// Mitsubishi GX Works2 project: PARKING   PLC: FX1S
// PARKING

PROGRAM MAIN
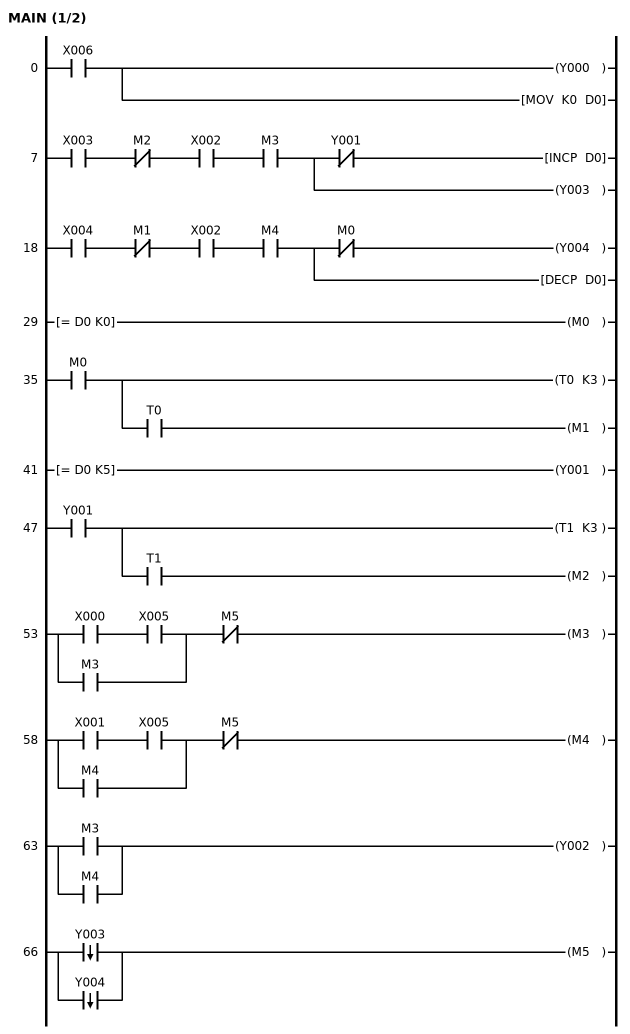
0     LD      X006
      OUT     Y000
      MOV     K0 D0
7     LD      X003
      ANI     M2
      AND     X002
      AND     M3
      MPS
      ANI     Y001
      INCP    D0
      MPP
      OUT     Y003
18    LD      X004
      ANI     M1
      AND     X002
      AND     M4
      MPS
      ANI     M0
      OUT     Y004
      MPP
      DECP    D0
29    LD=     D0 K0
      OUT     M0
35    LD      M0
      OUT     T0 K3
      AND     T0
      OUT     M1
41    LD=     D0 K5
      OUT     Y001
47    LD      Y001
      OUT     T1 K3
      AND     T1
      OUT     M2
53    LD      X000
      AND     X005
      OR      M3
      ANI     M5
      OUT     M3
58    LD      X001
      AND     X005
      OR      M4
      ANI     M5
      OUT     M4
63    LD      M3
      OR      M4
      OUT     Y002
66    LDF     Y003
      ORF     Y004
      OUT     M5
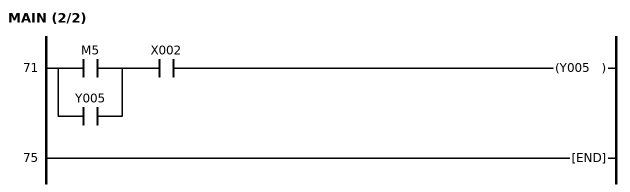
71    LD      M5
      OR      Y005
      AND     X002
      OUT     Y005
75    END
END_PROGRAM
